PROGRAM P_SunriseSunset
VAR
	bSunsetPulse		: BOOL;
	bSunrisePulse		: BOOL;

	rtSunset			: R_TRIG;
	ftSunset			: F_TRIG;
END_VAR

rtSunset(CLK:=bAdsSunIsDown, Q=>bSunsetPulse);
ftSunset(CLK:=bAdsSunIsDown, Q=>bSunrisePulse);

END_PROGRAM

(* stored: Version 1.1.0.1
   POU P_SunriseSunset: Id {8b91c887-ecff-4544-8b69-d0aeb75273c2}, SpecialFunc None *)
